{attribute 'qualified_only'}
TYPE ENU_DT0801EN03 :
(
	Signed_presentation := 0,
	Unsigned_presentation,
	Absolute_value_with_MSB_as_sign,
	Absolute_value
);
END_TYPE

(* stored: Version 1.1.0.1, ProductVersion 3.1.4024.6
   DUT ENU_DT0801EN03: Id {0cb8a9a3-ceb1-029a-2e57-649bb7a8dbad} *)
